(* IEC 61131-3 sources: A3br/, 3 files *)

(* ---- Types.typ ---- *)
(*//********************************************************************************
// Author:    Josh Polansky
// Created:   January 29, 2020
//*********************************************************************************)

TYPE
	A3brDigestAuthentication_typ : 	STRUCT
		count : USINT;
		password : STRING[80];
		userName : STRING[80];
		realm : STRING[1000];
		qop : STRING[30];
		nonce : STRING[100];
		opaque : STRING[100];
		cnonce : STRING[80];
		ABBCX : STRING[20];
		httpSession : STRING[100];
		nc : STRING[8];
		digest : STRING[32];
		requestId : STRING[200];
	END_STRUCT;
	A3brWebServiceCfg_typ : 	STRUCT
		hostname : STRING[80];
		port : UINT;
		username : STRING[80];
		password : STRING[80];
		maxSessions : USINT;
	END_STRUCT;
	A3brWebServiceRequest_typ : 	STRUCT
		self : UDINT;
		method : UDINT;
		successCallback : UDINT;
		errorCallback : UDINT;
		dataType : A3BR_REQ_DATA_TYPE_enum;
		uri : ARRAY[0..A3BR_STR_ROWS4]OF STRING[80];
		pBlock : UDINT;
		szBlock : UDINT;
		parameters : ARRAY[0..A3BR_MAI_REQUEST_PARS]OF A3brWebServiceRequestPar_typ;
	END_STRUCT;
	A3brWebServiceRequestPar_typ : 	STRUCT
		name : STRING[80];
		value : STRING[80];
	END_STRUCT;
	A3brWebServiceInternal_typ : 	STRUCT
		api : A3brWebServiceLink_typ;
		_reset : BOOL;
		session : ARRAY[0..2]OF A3brWebServiceSession_typ;
	END_STRUCT;
	A3brWebServiceSession_typ : 	STRUCT
		authTimeout : TON;
		authState : A3BR_AUTH_ST_enum;
		auth : A3brDigestAuthentication_typ;
		authRequest : A3brWebServiceAuthRequest_typ;
		connection : ARRAY[0..0]OF A3brWebServiceConnection_typ;
		reset : {REDUND_UNREPLICABLE} BOOL;
		connected : {REDUND_UNREPLICABLE} BOOL;
		activeConnections : {REDUND_UNREPLICABLE} UINT;
		inited : {REDUND_UNREPLICABLE} BOOL;
		error : USINT;
		errorID : USINT;
		errorString : STRING[80];
		_reset : {REDUND_UNREPLICABLE} BOOL;
	END_STRUCT;
	A3brWebServiceConnection_typ : 	STRUCT
		reqState : A3BR_REQUEST_ST_enum;
		httpClient : LLHttpClient;
		httpRequest : LLHttpRequest;
		reqData : ARRAY[0..A3BR_STR_ROWS20]OF STRING[80];
		resData : ARRAY[0..A3BR_STR_ROWS20]OF STRING[80];
		reqHeader : ARRAY[0..LLHTTP_MAI_NUM_HEADER_LINES]OF LLHttpHeaderField_typ;
		retries : UINT;
		responseTimeout : TON;
		currentRequest : A3brWebServiceRequest_typ;
		connected : BOOL;
		ping : TON;
		sent : BOOL;
		httpStatus : UINT;
	END_STRUCT;
	A3brWebServiceAuthRequest_typ : 	STRUCT
		uri : STRING[80];
		rawReqHeader : ARRAY[0..A3BR_STR_ROWS20]OF STRING[80];
		reqData : ARRAY[0..A3BR_STR_ROWS20]OF STRING[80];
		reqHeader : httpRequestHeader_t;
	END_STRUCT;
	A3brWebServiceLink_typ : 	STRUCT
		requestBuffer : Buffer_typ;
	END_STRUCT;
	A3brProgramControlInternal_typ : 	STRUCT
		done : BOOL;
		busy : BOOL;
		error : BOOL;
		errorID : UINT;
		errorString : STRING[80];
		_loadProgram : BOOL;
		_loadModule : BOOL;
	END_STRUCT;
	A3brControlInternal_typ : 	STRUCT
		done : BOOL;
		busy : BOOL;
		error : BOOL;
		errorID : UINT;
		errorString : STRING[80];
		_powerOn : BOOL;
		_powerOff : BOOL;
		_start : BOOL;
		_stop : BOOL;
		_continue : BOOL;
		_reset : BOOL;
		_requestMastership : BOOL;
		_releaseMastership : BOOL;
	END_STRUCT;
	A3brGetStateInternal_typ : 	STRUCT
		done : BOOL;
		busy : BOOL;
		error : BOOL;
		successCount : UDINT;
		errorID : UINT;
		errorString : STRING[80];
		oldUpdate : BOOL;
		update : BOOL;
		updateTimer : TON;
	END_STRUCT;
	A3brSetSymbolInternal_typ : 	STRUCT
		done : BOOL;
		busy : BOOL;
		error : BOOL;
		errorID : UINT;
		errorString : STRING[80];
		_cmd : BOOL;
	END_STRUCT;
	A3brSetIOInternal_typ : 	STRUCT
		done : BOOL;
		busy : BOOL;
		error : BOOL;
		errorID : UINT;
		errorString : STRING[80];
		_cmd : BOOL;
	END_STRUCT;
	A3brIOWatchIOInternal_typ : 	STRUCT
		oValue : INT;
		value : INT;
		pValue : REFERENCE TO INT;
		busy : BOOL;
		error : BOOL;
		errorID : UINT;
		errorString : STRING[80];
	END_STRUCT;
	A3brIOWatchInternal_typ : 	STRUCT
		readIndex : USINT;
		refresh : TON;
		pIO : UDINT;
	END_STRUCT;
	A3brGetSymbolInternal_typ : 	STRUCT
		done : BOOL;
		busy : BOOL;
		error : BOOL;
		errorID : UINT;
		errorString : STRING[80];
		_cmd : BOOL;
		data : ARRAY[0..79]OF USINT;
	END_STRUCT;
	A3brGetIOInternal_typ : 	STRUCT
		done : BOOL;
		busy : BOOL;
		error : BOOL;
		errorID : UINT;
		errorString : STRING[80];
		_cmd : BOOL;
	END_STRUCT;
	A3BR_AUTH_ST_enum :
		(
		A3BR_AUTH_ST_INIT := 0,
		A3BR_AUTH_ST_WAIT_FOR_SERVER := 1,
		A3BR_AUTH_ST_AUTHENTICATE := 2,
		A3BR_AUTH_ST_AUTHENTICATE_SENT := 3,
		A3BR_AUTH_ST_READY := 4,
		A3BR_AUTH_ST_ERROR := 500
		);
	A3BR_REQUEST_ST_enum :
		(
		A3BR_REQUEST_ST_IDLE := 0,
		A3BR_REQUEST_ST_GENERATE_STRING := 1,
		A3BR_REQUEST_ST_SEND := 2,
		A3BR_REQUEST_ST_PROCESS_RESPONSE := 3
		);
	A3BR_VAR_TYPE_enum :
		(
		A3BR_VAR_TYPE_BOOL,
		A3BR_VAR_TYPE_INT,
		A3BR_VAR_TYPE_REAL,
		A3BR_VAR_TYPE_STRING
		);
END_TYPE

(*States*)

TYPE
	A3BR_RAPID_EXEC_ST_enum :
		(
		A3BR_RAPID_EXEC_ST_UNDEFINED,
		A3BR_RAPID_EXEC_ST_RUNNING, (*ABB constant "running"*)
		A3BR_RAPID_EXEC_ST_STOPPED (*ABB constant "stopped"*)
		);
	A3BR_RAPID_CYCLE_ST_enum :
		(
		A3BR_RAPID_CYCLE_ST_UNDEFINED,
		A3BR_RAPID_CYCLE_ST_FOREVER, (*ABB constant "forever": this repeats the program forever*)
		A3BR_RAPID_CYCLE_ST_ASIS, (*ABB constant "asis": this keeps the current cycle state on the IRC5*)
		A3BR_RAPID_CYCLE_ST_ONCE, (*ABB constant "once": this runs the program a single time*)
		A3BR_RAPID_CYCLE_ST_ONCEDONE (*ABB constant "oncedone"*)
		);
	A3BR_CTRL_ST_enum :
		(
		A3BR_CTRL_ST_UNDEFINED,
		A3BR_CTRL_ST_INIT, (*ABB constant "init": The robot is starting up. It will shift to state motors off when it has started.*)
		A3BR_CTRL_ST_ON, (*ABB constant "motoron": The robot is ready to move, either by jogging or by running programs.*)
		A3BR_CTRL_ST_OFF, (*ABB constant "motoroff": The robot is in a standby state where there is no power to the robot's motors. The state has to be shifted to motors on before the robot can move.*)
		A3BR_CTRL_ST_GUARDSTOP, (*ABB constant "guardstop": The robot is stopped because the safety runchain is opened. For instance, a door to the robot's cell might be open.*)
		A3BR_CTRL_ST_ESTOP, (*ABB constant "emergencystop": The robot is stopped because emergency stop was activated.*)
		A3BR_CTRL_ST_ESTOP_RESET, (*ABB constant "emergencystopreset": The robot is ready to leave emergency stop state. The emergency stop is no longer activated, but the state transition isn't yet confirmed.*)
		A3BR_CTRL_ST_SYS_FAIL (*ABB constant "sysfail": The robot is in a system failure state. Restart required.*)
		);
	A3BR_OP_MODE_enum :
		(
		A3BR_OP_MODE_UNDEFINED, (*ABB constant "UNDEF": Undefined*)
		A3BR_OP_MODE_INIT, (*ABB constant "INIT": State init*)
		A3BR_OP_MODE_AUTO_CHANGE_REQ, (*ABB constant "AUTO_CH": State change request for automatic mode*)
		A3BR_OP_MODE_MANUAL_CHANGE_REQ, (*ABB constant "MANF_CH": State change request for manual mode & full speed*)
		A3BR_OP_MODE_MANUAL_LOW_SPEED, (*ABB constant "MANR": State manual mode & reduced speed*)
		A3BR_OP_MODE_MANUAL_FULL_SPEED, (*ABB constant "MANF": State manual mode & full speed*)
		A3BR_OP_MODE_AUTO (*ABB constant "AUTO": State automatic mode*)
		);
	A3BR_ERR_enum :
		(
		A3BR_ERR_INVALID_IDENT := 56000,
		A3BR_ERR_AUTH_TIMEOUT := 56001,
		A3BR_ERR_RESPONSE_TIMEOUT := 56002,
		A3BR_ERR_HTTP_ERROR := 56003,
		A3BR_ERR_INSUFFICIENT_SIGNALS := 56004,
		A3BR_ERR_INVALID_CYCLE := 56005,
		A3BR_ERR_INVALID_NAME := 56006,
		A3BR_ERR_INVALID_DATA_ADDRESS := 56007,
		A3BR_ERR_INVALID_DATA_SIZE := 56008
		);
	A3BR_REQ_DATA_TYPE_enum :
		(
		A3BR_REQ_DATA_TYPE_PARS := 0,
		A3BR_REQ_DATA_TYPE_BLOCK := 1
		);
	A3BR_GET_STATE_MODE_enum :
		(
		A3BR_GET_STATE_MODE_SINGLE,
		A3BR_GET_STATE_MODE_CONTINUOUS
		);
END_TYPE

(* ---- a3br.fun ---- *)
(*//********************************************************************************
// Author:    Josh Polansky
// Created:   January 29, 2020
//*********************************************************************************)

FUNCTION_BLOCK A3brWebService (*Establish the initial connection to the IRC, and handle channeling of all HTTP traffic back and forth.*)
	VAR_INPUT
		enable : BOOL;
		reset : BOOL;
		configuration : A3brWebServiceCfg_typ;
	END_VAR
	VAR_OUTPUT
		ident : UDINT;
		connected : BOOL;
		activeSessions : UINT;
		activeConnections : UINT;
		error : BOOL;
		errorID : UINT;
		errorString : STRING[80];
	END_VAR
	VAR
		internal : A3brWebServiceInternal_typ;
	END_VAR
END_FUNCTION_BLOCK

FUNCTION_BLOCK A3brControl (*Send high level commands to the IRC to control robot execution state.*)
	VAR_INPUT
		ident : UDINT;
		powerOn : BOOL;
		powerOff : BOOL;
		start : BOOL;
		stop : BOOL;
		reset : BOOL;
		requestMastership : BOOL;
		releaseMastership : BOOL;
		cycle : A3BR_RAPID_CYCLE_ST_enum;
	END_VAR
	VAR_OUTPUT
		busy : BOOL;
		done : BOOL;
		error : BOOL;
		errorID : UINT;
		errorString : STRING[80];
	END_VAR
	VAR
		internal : A3brControlInternal_typ;
	END_VAR
END_FUNCTION_BLOCK

FUNCTION_BLOCK A3brProgramControl (*Send high level commands to the IRC to control robot execution state.*)
	VAR_INPUT
		ident : UDINT;
		loadProgram : BOOL;
		loadModule : BOOL;
		pProgramName : {REDUND_UNREPLICABLE} UDINT;
		pModuleName : UDINT;
		pTaskName : UDINT;
		pData : UDINT;
		szData : UDINT;
	END_VAR
	VAR_OUTPUT
		busy : BOOL;
		done : BOOL;
		error : BOOL;
		errorID : UINT;
		errorString : STRING[80];
	END_VAR
	VAR
		internal : A3brProgramControlInternal_typ;
	END_VAR
END_FUNCTION_BLOCK

FUNCTION_BLOCK A3brSetIO (*Write a value to an IO signal on the IRC.*)
	VAR_INPUT
		ident : UDINT;
		execute : BOOL;
		pSignal : REFERENCE TO STRING[A3BR_IO_STR_LEN];
		mode : {REDUND_UNREPLICABLE} UDINT; (*not implemented*)
		value : {REDUND_UNREPLICABLE} INT; (*not implemented*)
		delay : {REDUND_UNREPLICABLE} UDINT; (*not implemented*)
		pulses : {REDUND_UNREPLICABLE} UDINT; (*not implemented*)
		activePulse : {REDUND_UNREPLICABLE} UDINT; (*not implemented*)
		passivePulse : {REDUND_UNREPLICABLE} UDINT; (*not implemented*)
	END_VAR
	VAR_OUTPUT
		busy : BOOL;
		done : BOOL;
		error : BOOL;
		errorID : UINT;
		errorString : STRING[80];
	END_VAR
	VAR
		internal : A3brSetIOInternal_typ;
	END_VAR
END_FUNCTION_BLOCK

FUNCTION_BLOCK A3brGetIO (*Read the value of an IO signal from the IRC.*)
	VAR_INPUT
		ident : UDINT;
		execute : BOOL;
		pSignal : REFERENCE TO STRING[A3BR_IO_STR_LEN];
	END_VAR
	VAR_OUTPUT
		value : INT;
		busy : BOOL;
		done : BOOL;
		error : BOOL;
		errorID : UINT;
		errorString : STRING[80];
	END_VAR
	VAR
		internal : A3brGetIOInternal_typ;
	END_VAR
END_FUNCTION_BLOCK

FUNCTION_BLOCK A3brSetSymbol (*Write a value to an IO signal on the IRC.*)
	VAR_INPUT
		ident : UDINT;
		execute : BOOL;
		pSignal : REFERENCE TO STRING[A3BR_SYMBOL_STR_LEN];
		pValue : UDINT;
		szValue : UDINT;
		typeValue : A3BR_VAR_TYPE_enum;
		mode : {REDUND_UNREPLICABLE} UDINT; (*not implemented*)
		delay : {REDUND_UNREPLICABLE} UDINT; (*not implemented*)
		pulses : {REDUND_UNREPLICABLE} UDINT; (*not implemented*)
		activePulse : {REDUND_UNREPLICABLE} UDINT; (*not implemented*)
		passivePulse : {REDUND_UNREPLICABLE} UDINT; (*not implemented*)
	END_VAR
	VAR_OUTPUT
		busy : BOOL;
		done : BOOL;
		error : BOOL;
		errorID : UINT;
		errorString : STRING[80];
	END_VAR
	VAR
		internal : A3brSetSymbolInternal_typ;
	END_VAR
END_FUNCTION_BLOCK

FUNCTION_BLOCK A3brGetSymbol (*Read the value of an IO signal from the IRC.*)
	VAR_INPUT
		ident : UDINT;
		execute : BOOL;
		pSignal : REFERENCE TO STRING[A3BR_SYMBOL_STR_LEN];
		pValue : UDINT;
		szValue : UDINT;
		typeValue : A3BR_VAR_TYPE_enum;
	END_VAR
	VAR_OUTPUT
		busy : BOOL;
		done : BOOL;
		error : BOOL;
		errorID : UINT;
		errorString : STRING[80];
	END_VAR
	VAR
		internal : A3brGetSymbolInternal_typ;
	END_VAR
END_FUNCTION_BLOCK

FUNCTION_BLOCK A3brGetState (*Read high level state information from the IRC.*)
	VAR_INPUT
		ident : UDINT;
		enable : BOOL;
		mode : A3BR_GET_STATE_MODE_enum;
		cycleTime : UDINT;
	END_VAR
	VAR_OUTPUT
		rapidExecutionState : A3BR_RAPID_EXEC_ST_enum;
		rapidCycleState : A3BR_RAPID_CYCLE_ST_enum;
		controlState : A3BR_CTRL_ST_enum;
		operationalMode : A3BR_OP_MODE_enum;
		busy : BOOL;
		done : BOOL;
		successCount : UDINT;
		error : BOOL;
		errorID : UINT;
		errorString : STRING[80];
	END_VAR
	VAR
		internal : A3brGetStateInternal_typ;
	END_VAR
END_FUNCTION_BLOCK

FUNCTION_BLOCK A3brIOWatch (*Set up cyclic read/write watch for a list of IO signals on the IRC. *)
	VAR_INPUT
		enable : BOOL;
		ident : UDINT;
		pSignals : REFERENCE TO ARRAY[0..0] OF STRING[A3BR_IO_STR_LEN];
		pValues : REFERENCE TO INT;
		numSignals : USINT;
		maxCycleReads : USINT;
		refresh : TIME;
	END_VAR
	VAR_OUTPUT
		error : BOOL;
		errorID : UINT;
		errorString : STRING[80];
	END_VAR
	VAR
		internal : A3brIOWatchInternal_typ;
	END_VAR
END_FUNCTION_BLOCK

FUNCTION A3brRapidExec2String : UINT
	VAR_INPUT
		rapidExec : UINT;
		pString : UDINT;
	END_VAR
END_FUNCTION

FUNCTION A3brRapidCycle2String : UINT
	VAR_INPUT
		rapidCycle : UINT;
		pString : UDINT;
	END_VAR
END_FUNCTION

FUNCTION A3brCtrlState2String : UINT
	VAR_INPUT
		ctrlState : UINT;
		pString : UDINT;
	END_VAR
END_FUNCTION

FUNCTION A3brOpMode2String : UINT
	VAR_INPUT
		opMode : UINT;
		pString : UDINT;
	END_VAR
END_FUNCTION

(* ---- Constants.var ---- *)
(*//********************************************************************************
// Author:    Josh Polansky
// Created:   January 29, 2020
//*********************************************************************************)
VAR CONSTANT
	A3BR_MAI_REQUEST_PARS : UINT := 19;
	A3BR_IO_STR_LEN : UINT := 80;
	A3BR_SYMBOL_STR_LEN : UINT := 80;
	A3BR_STR_ROWS4 : UINT := 19; (*	*)
	A3BR_STR_ROWS20 : UINT := 19; (*	*)
END_VAR
